(* CoDeSys 2.3 export: HEATPLACEE.EXP *)

(* Data type in BathFB *)
(*расположение нагревателя*)
TYPE HeatPlaceE :
(
    US_1,
    US_2,
    Wash
);
END_TYPE
